{attribute 'pack_mode' := '1'}
TYPE TProductionCmd :
STRUCT
	TRequestSample		: TManButton;
	TAutoSampling		: TAutoSampling;
END_STRUCT
END_TYPE

(* stored: Version 1.1.0.1, ProductVersion 3.1.4022.12
   DUT TProductionCmd: Id {61b378f8-b6b0-4d7d-83b9-776e005126aa} *)
